// SIMATIC S7-200 SMART project (STEP 7-Micro/WIN SMART), CPU SR40

SYMBOL_TABLE Table 1
Timer_Run        M1.4     // Allow movement
Time_Short_Signal T210
Greate_Min_bit   M4.0     // Allow buzer if timer great 1 min
Timeout_Fail     T200
Time_Signal      T220
END_SYMBOL_TABLE

SYMBOL_TABLE System Symbols
Always_On        SM0.0    // Always ON
First_Scan_On    SM0.1    // ON for the first scan cycle only
Clock_1s         SM0.5    // Clock pulse that is ON for 0.5 s, OFF for 0.5 s, for a duty cycle time of 1 s.
END_SYMBOL_TABLE

ORGANIZATION_BLOCK Program_Block:OB1
TITLE=Program Comments
BEGIN
Network 1
// Network Comment
LD     First_Scan_On:SM0.1
LD     T101
NOT
A      M1.7
OLD
=      M1.7
TON    T101, +20
Network 2
LD     T101
R      CPU_Output0:Q0.0, 16
R      M0.0, 16
R      T37, 5
Network 3
// (network saved uncompiled; FBD cells follow)
// row 1: c3 [S1 SR M0.0 CPU_Input7:I0.7 R:=power@row2, OUT=>power]  c4 -- v  c5 --  c6 [= CPU_Output11:Q1.3 ]
// row 2: c1 [OR CPU_Input6:I0.6 V0.4 ]  c2 --  c3 [box]  c4 ^v
// row 3: c1 [box]  c4 ^v  c5 --  c6 [R M1.2 N:=8]
// row 4: c4 ^v  c6 [box]
// row 5: c4 ^v
// row 6: c4 ^v  c5 --  c6 [= V11.1 ]
// row 7: c4 ^v  c6 [MOV_W ]
// row 8: c4 ^  c5 --  c6 [ EN:=power@row8, IN:=+2, ENO=>V?0, OUT=>MW8]
// row 9: c6 [box]
Network 4
// (network saved uncompiled; FBD cells follow)
// row 1: c3 [SR M0.1 S1:=CPU_Input10:I1.2, R:=power@row2, OUT=>power]  c4 -- v  c5 --  c6 [= V11.0 ]
// row 2: c1 [OR CPU_Input6:I0.6 V0.4 ]  c2 --  c3 [box]  c4 ^v  c6 [MOV_W ]
// row 3: c1 [box]  c4 ^  c5 --  c6 [ EN:=power@row3, IN:=+2, ENO=>V?0, OUT=>MW8]
// row 4: c6 [box]
Network 5
LDN    M0.2
TON    T37, +50
Network 6
LDN    M0.3
TON    T38, +50
Network 7
LD     M0.4
O      M0.5
LPS
AN     V0.1
AN     M0.3
A      T38
=      M0.2
LPP
A      V0.1
AN     M0.2
A      T37
=      M0.3
Network 8
LDN    V0.0
=      M0.5
Network 9
LD     V0.0
=      M0.4
Network 10
LD     CPU_Input1:I0.1
LD     CPU_Input0:I0.0
A      M0.5
NOT
LPS
A      M0.6
=      M0.6
LPP
ALD
O      M0.6
=      M0.6
=      CPU_Output9:Q1.1
Network 11
// (network saved uncompiled; FBD cells follow)
// row 1: c1 [OR CPU_Input6:I0.6 V0.4 ]  c2 --  c3 [RS M0.7 S:=power@row1, R1:=power@row3, OUT=>power]  c4 -- v  c5 --  c6 [= CPU_Output10:Q1.2 ]
// row 2: c1 [box]  c3 [box]  c4 ^v  c6 [MOV_W ]
// row 3: c1 [OR M0.1 CPU_Input7:I0.7 ]  c2 --  c3 [box]  c4 ^  c5 --  c6 [ EN:=power@row3, IN:=+1, ENO=>V?0, OUT=>MW8]
// row 4: c1 [box]  c6 [box]
Network 12
LD     V0.2
LD     V0.3
NOT
LPS
A      M1.0
=      M1.0
LPP
ALD
O      M1.0
=      M1.0
=      CPU_Output0:Q0.0
Network 13
// (network saved uncompiled; FBD cells follow)
// row 1: c2 [AND CPU_Input0:I0.0 M0.5 ]  c3 --  c4 [RS M1.1 S:=power@row1, R1:=power@row5, OUT=>V?0]
// row 2: c2 [box]  c4 [box]
// row 3: c1 [<>I VW400 +0 ]  c2 [box]  c4 [box]
// row 4: c1 [box]  c4 [box]
// row 5: c2 [OR CPU_Input1:I0.1 M0.1 M0.0 ]  c3 --  c4 [box]
// row 6: c2 [box]
// row 7: c2 [box]
Network 14
LD     M1.1
TON    T39, +20
Network 15
// (network saved uncompiled; FBD cells follow)
// row 1: c1 [AND T39 M0.5 M2.1 ]  c2 --  c3 [RS M1.2 S:=power@row1, R1:=C0, OUT=>V?0]
// row 2: c1 [box]  c3 [box]
// row 3: c1 [box]
Network 16
LD     Always_On:SM0.0
AW=    C1, +0
EU
=      M2.1
Network 17
// (network saved uncompiled; FBD cells follow)
// row 1: c1 [AND M0.4 CPU_Input0:I0.0 ]  c2 --  c3 [RS M1.3 S:=power@row1, R1:=C0, OUT=>V?0]
// row 2: c1 [box]  c3 [box]
Network 18
LD     CPU_Input2:I0.2
ED
AN     CPU_Output14:Q1.6
LD     CPU_Input2:I0.2
ED
O      First_Scan_On:SM0.1
A      CPU_Output14:Q1.6
NOT
A      M1.6
OLD
=      M1.6
=      CPU_Output14:Q1.6
Network 19
// (network saved uncompiled; FBD cells follow)
// row 1: c1 [AND M0.5 M1.1 ]  c2 --  c3 [P ]  c4 [OR ]  c5 --  c6 [RS Timer_Run:M1.4 S:=power@row1, R1:=power@row5, OUT=>V?0]
// row 2: c1 [box]  c4 [box]  c6 [box]
// row 3: c1 [AND M0.5 C0 ]  c2 --  c3 [P ]  c4 [box]  c6 [box]
// row 4: c1 [box]  c6 [box]
// row 5: c1 [AND M0.5 M0.6 ]  c2 --  c3 [P ]  c4 [OR ]  c5 --  c6 [box]
// row 6: c1 [box]  c4 [box]
// row 7: c1 [AND M0.5 M0.0 ]  c2 --  c3 [P ]  c4 [box]
// row 8: c1 [box]  c4 [box]
// row 9: c1 [AND M0.5 M0.1 ]  c2 --  c3 [P ]  c4 [box]
// row 10: c1 [box]  c4 [box]
// row 11: c1 [AND M0.5 M1.2 ]  c2 --  c3 [P ]  c4 [box]
// row 12: c1 [box]
Network 20
LD     Timer_Run:M1.4
A      Clock_1s:SM0.5
AN     M1.6
LD     Timer_Run:M1.4
EU
CTD    C1, VW400
Network 21
LD     Always_On:SM0.0
CALL   时间处理程序:SBR1
Network 22
LD     CPU_Input9:I1.1
EU
LD     C0
CTU    C0, +4
Network 23
LD     C0
=      M1.5
Network 24
// set bit allow move
LD     M1.3
O      M1.2
=      Motor_on:Q0.4
Network 25
LD     M1.2
O      M1.3
LPS
AN     CPU_Output6:Q0.6
AN     M1.6
AN     CPU_Input11:I1.3
A      M0.2
=      CPU_Output5:Q0.5
LPP
AN     CPU_Output5:Q0.5
AN     M1.6
AN     CPU_Input12:I1.4
A      M0.3
=      CPU_Output6:Q0.6
Network 26
LD     T39
LD     CPU_Output5:Q0.5
O      CPU_Output6:Q0.6
ALD
A      M0.5
LD     CPU_Output5:Q0.5
O      CPU_Output6:Q0.6
A      M1.3
LD     T39
AN     M1.2
OLD
AN     Clock_1s:SM0.5
OLD
=      CPU_Output8:Q1.0
Network 27
LD     M0.1
O      M0.0
=      Buzer_On:Q1.5
Network 28
LD     Motor_on:Q0.4
AN     Timeout_Fail:T200
TON    Timeout_Fail:T200, +200
Network 29
LD     M1.0
=      V0.5
Network 30
LDN    M1.0
=      V0.6
Network 31
// (network saved uncompiled; FBD cells follow)
// row 0: c1 [READ_RTC ]
// row 1: c1 [ EN:=Clock_1s:SM0.5, T:=VB1700, ENO=>V?0]
// row 2: c1 [box]
Network 32
LD     Always_On:SM0.0
CALL   通迅:SBR0
Network 33
LD     M4.1
O      M4.2
=      Buzer_On:Q1.5
Network 34
// Signale fail
// (network saved uncompiled; FBD cells follow)
// row 1: c1 [AND Motor_on:Q0.4 Timeout_Fail:T200 ]  c2 --  c3 [RS M4.1 S:=power@row1, R1:=Time_Short_Signal:T210, OUT=>V?0]
// row 2: c1 [box]  c3 [box]
END_ORGANIZATION_BLOCK

SUBROUTINE_BLOCK 通迅:SBR0
TITLE=Subroutine Comments
BEGIN
Network 1
// Network Comment
LD     Always_On:SM0.0
=      L60.0
LD     Always_On:SM0.0
=      L63.7
LD     L60.0
CALL   MBUS_CTRL:SBR2, L63.7, 9600, 0, 1, +1000, M10.0, MB20
Network 2
LD     Always_On:SM0.0
=      L60.0
LD     Clock_1s:SM0.5
EU
LD     M13.0
EU
OLD
=      L63.7
LD     L60.0
CALL   MBUS_MSG:SBR3, L63.7, 3, 1, 40002, +1, &VB300, M10.1, MB21
Network 3
LD     M10.1
R      M13.0, 1
S      M13.1, 1
Network 4
LD     M30.0
R      M10.1, 1
Network 5
// Sound if timer count > min
LD     M4.2
TON    Time_Signal:T220, +7
Network 6
// Sound if fail
LD     M4.1
TON    Time_Short_Signal:T210, +5
Network 7
// Signal if great min
// (network saved uncompiled; FBD cells follow)
// row 1: c1 [==I C1 +7 ]  c2 [AND Greate_Min_bit:M4.0 M4.3 ]  c3 --  c4 [RS M4.2 S:=power@row1, R1:=Time_Signal:T220, OUT=>V?0]
// row 2: c1 [box]  c2 [box]  c4 [box]
// row 3: c2 [box]
// row 4: c2 [box]
Network 8
// Once signal for cicle
// (network saved uncompiled; FBD cells follow)
// row 1: c1 [RS M4.3 S:=M4.2, R1:=C0, OUT=>V?0]
// row 2: c1 [box]
END_SUBROUTINE_BLOCK

SUBROUTINE_BLOCK 时间处理程序:SBR1
TITLE=
BEGIN
Network 1
// (network saved uncompiled; FBD cells follow)
// row 0: c1 [MOV_W ]
// row 1: c1 [ EN:=Always_On:SM0.0, IN:=C1, ENO=>V?0, OUT=>VW500]
// row 2: c1 [box]
Network 2
// (network saved uncompiled; FBD cells follow)
// row 0: c3 [MOV_W ]
// row 1: c1 [<>I VW400 +0 ]  c2 --  c3 [ EN:=power@row1, IN:=VW400, ENO=>V?0, OUT=>VW22]
// row 2: c1 [box]  c3 [box]
Network 3
// (network saved uncompiled; FBD cells follow)
// row 0: c3 [DIV ]
// row 1: c1 [<>I VW400 +0 ]  c2 --  c3 [ EN:=power@row1, IN1:=VW22, IN2:=+60, ENO=>V?0, OUT=>VD16]
// row 2: c1 [box]  c3 [box]
// row 3: c3 [box]
Network 4
// (network saved uncompiled; FBD cells follow)
// row 0: c4 [DIV ]
// row 1: c2 [AND Always_On:SM0.0 ]  c3 --  c4 [ EN:=power@row1, IN1:=VW500, IN2:=+3600, ENO=>V?0, OUT=>VD100]
// row 2: c1 [>=I VW500 +3600 ]  c2 [box]  c4 [box]
// row 3: c1 [box]  c4 [box]
Network 5
// (network saved uncompiled; FBD cells follow)
// row 0: c4 [MOV_DW ]
// row 1: c2 [AND Always_On:SM0.0 ]  c3 --  c4 [ EN:=power@row1, IN:=+0, ENO=>V?0, OUT=>VD100]
// row 2: c1 [<I VW500 +3600 ]  c2 [box]  c4 [box]
// row 3: c1 [box]
Network 6
// (network saved uncompiled; FBD cells follow)
// row 0: c4 [DIV ]
// row 1: c2 [AND Always_On:SM0.0 ]  c3 --  c4 [ EN:=power@row1, IN1:=VW500, IN2:=+60, ENO=>V?0, OUT=>VD200]
// row 2: c1 [>I VW500 +59 ]  c2 [box]  c4 [box]
// row 3: c1 [box]  c2 [box]  c4 [box]
// row 4: c1 [<I VW500 +3600 ]  c2 [box]
// row 5: c1 [box]
Network 7
LD     Always_On:SM0.0
AW>    VW500, +59
AW<    VW500, +3600
=      M2.2
Network 8
// (network saved uncompiled; FBD cells follow)
// row 0: c4 [DIV ]
// row 1: c2 [AND Always_On:SM0.0 M2.2 ]  c3 --  c4 [ EN:=power@row1, IN1:=VW100, IN2:=+60, ENO=>V?0, OUT=>VD200]
// row 2: c1 [>=I VW100 +60 ]  c2 [box]  c4 [box]
// row 3: c1 [box]  c2 [box]  c4 [box]
// row 4: c2 [box]
Network 9
// (network saved uncompiled; FBD cells follow)
// row 0: c4 [MOV_DW ]
// row 1: c2 [AND Always_On:SM0.0 ]  c3 --  c4 [ EN:=power@row1, IN:=+0, ENO=>V?0, OUT=>VD200]
// row 2: c1 [<I VW500 +60 ]  c2 [box]  c4 [box]
// row 3: c1 [box]
Network 10
// (network saved uncompiled; FBD cells follow)
// row 0: c4 [MOV_W ]
// row 1: c2 [AND Always_On:SM0.0 ]  c3 --  c4 [ EN:=power@row1, IN:=VW500, ENO=>V?0, OUT=>VW20]
// row 2: c1 [<=I VW500 +59 ]  c2 [box]  c4 [box]
// row 3: c1 [box]
Network 11
LD     Always_On:SM0.0
AW<=   VW500, +59
=      M2.0
Network 12
// (network saved uncompiled; FBD cells follow)
// row 0: c4 [MOV_W ]
// row 1: c2 [AND Always_On:SM0.0 M2.0 ]  c3 --  c4 [ EN:=power@row1, IN:=VW200, ENO=>V?0, OUT=>VW20]
// row 2: c1 [<=I VW200 +59 ]  c2 [box]  c4 [box]
// row 3: c1 [box]  c2 [box]
// row 4: c2 [box]
Network 13
LD     Always_On:SM0.0
AW<=   VW200, +59
=      M2.3
Network 14
// (network saved uncompiled; FBD cells follow)
// row 0: c4 [MOV_W ]
// row 1: c2 [AND Always_On:SM0.0 M2.0 M2.3 ]  c3 --  c4 [ EN:=power@row1, IN:=VW100, ENO=>V?0, OUT=>VW20]
// row 2: c1 [<=I VW100 +59 ]  c2 [box]  c4 [box]
// row 3: c1 [box]  c2 [box]
// row 4: c2 [box]
// row 5: c2 [box]
Network 15
// (network saved uncompiled; FBD cells follow)
// row 0: c1 [MOV_W ]
// row 1: c1 [ EN:=Always_On:SM0.0, IN:=VW202, ENO=>V?0, OUT=>VW26]
// row 2: c1 [box]
Network 16
// (network saved uncompiled; FBD cells follow)
// row 0: c1 [MOV_W ]
// row 1: c1 [ EN:=Always_On:SM0.0, IN:=VW102, ENO=>V?0, OUT=>VW24]
// row 2: c1 [box]
Network 17
// (network saved uncompiled; FBD cells follow)
// row 0: c1 [MOV_W ]
// row 1: c1 [ EN:=Always_On:SM0.0, IN:=VW500, ENO=>V?0, OUT=>VW300]
// row 2: c1 [box]
Network 18
// Count timer greate min 
// (network saved uncompiled; FBD cells follow)
// row 1: c1 [>I VW500 +59 ]  c2 --  c3 [RS Greate_Min_bit:M4.0 S:=power@row1, R1:=Motor_on:Q0.4, OUT=>V?0]
// row 2: c1 [box]  c3 [box]
END_SUBROUTINE_BLOCK

// SBR2: protected block, not included

// SBR3: protected block, not included

// SBR4: protected block, not included

// INT1: protected block, not included
